# EPICS autosave request: ESP300/iocBoot/ioc_esp_bmb/auto_settings.req
file "XFM_motor_settings.req",        P=XF:04BMB-OP:, M=MBV-Cam:Y:Mtr
